// TIA Portal V19 export
TYPE "LEXCHANGETRAY_typePc_controlPar"
// stored: Access Published
   STRUCT
      cellSize : Int;   // cellSize
   END_STRUCT;
END_TYPE
